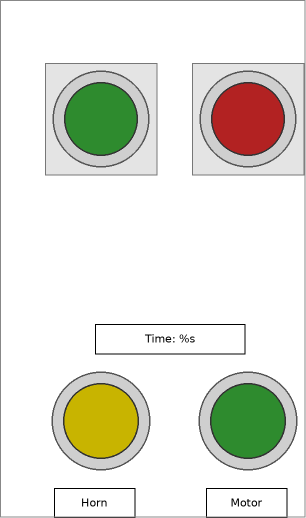
VISUALIZATION Visualization  // 306x518
    PushSwitch (43,63 116x112), variable: MAIN.bStartButton, behaviour: TOGGLE, style: Switch-PushSwitch-Green
    PushSwitch (190,63 116x112), variable: MAIN.bStopButton, behaviour: TOGGLE, style: Switch-PushSwitch-Red
    Lamp1 (43,364 116x114), variable: MAIN.bHorn, style: Lamp-Lamp1-Yellow
    Lamp1 (190,364 116x114), variable: MAIN.bMotor, style: Lamp-Lamp1-Green
    Rectangle (95,324 150x30), "Time: %s", text variable: MAIN.fbStartupTimer.ET
    Rectangle (54,488 81x30), "Horn", text variable: MAIN.fbStartupTimer.ET
    Rectangle (206,488 81x30), "Motor", text variable: MAIN.fbStartupTimer.ET
END_VISUALIZATION

(* stored: Version 1.1.0.1
   Visu Visualization: Id {65f3f850-489f-4d15-9ff9-d9d0cb0b4b68} *)
